FUNCTION_BLOCK AxisWriteParameter
VAR_INPUT
	Execute_:BOOL;
	Begin_Position:INT;
	End_Position:INT;
END_VAR
VAR_OUTPUT
END_VAR
VAR
	Write_Bool_Start	:	MC_WriteBoolParameter;
	Write_Bool_End 	:	MC_WriteBoolParameter;
	Write_Start :	MC_WriteParameter;
	Write_End :	MC_WriteParameter;
END_VAR

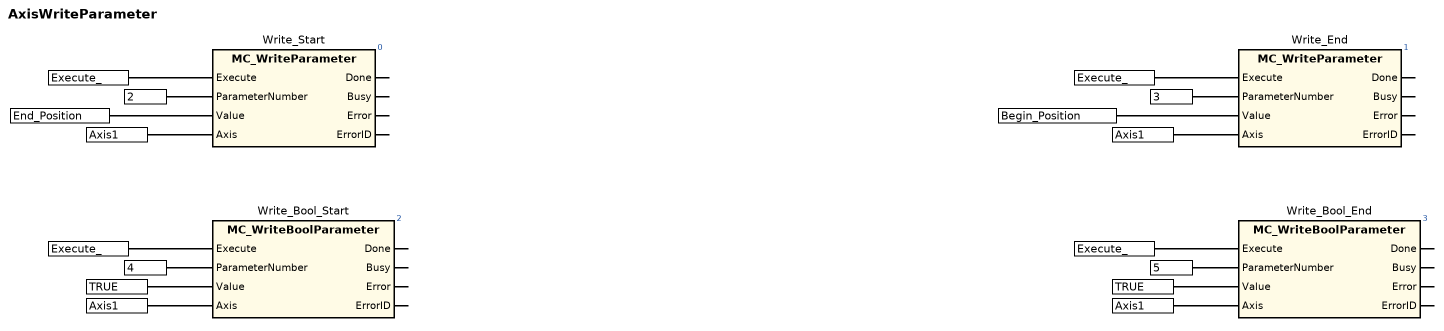
Write_Start(Execute := Execute_, ParameterNumber := 2, Value := End_Position, Axis := Axis1); // MC_WriteParameter
Write_End(Execute := Execute_, ParameterNumber := 3, Value := Begin_Position, Axis := Axis1); // MC_WriteParameter
Write_Bool_Start(Execute := Execute_, ParameterNumber := 4, Value := TRUE, Axis := Axis1); // MC_WriteBoolParameter
Write_Bool_End(Execute := Execute_, ParameterNumber := 5, Value := TRUE, Axis := Axis1); // MC_WriteBoolParameter

END_FUNCTION_BLOCK

(* stored: Version 1.1.0.1, ProductVersion 3.1.4024.12
   POU AxisWriteParameter: Id {4be5469a-3bff-4e92-945b-262c576c0b5e}, SpecialFunc None *)
